SUBAPPLICATION Uebung_072c (* GBSD auf UT ausgeben *)
  (* Standard: 61499-2 *)
  (* Version 1.0, 2023-10-23, franz *)
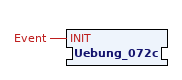
  EVENT_INPUT
    INIT;
  END_EVENT
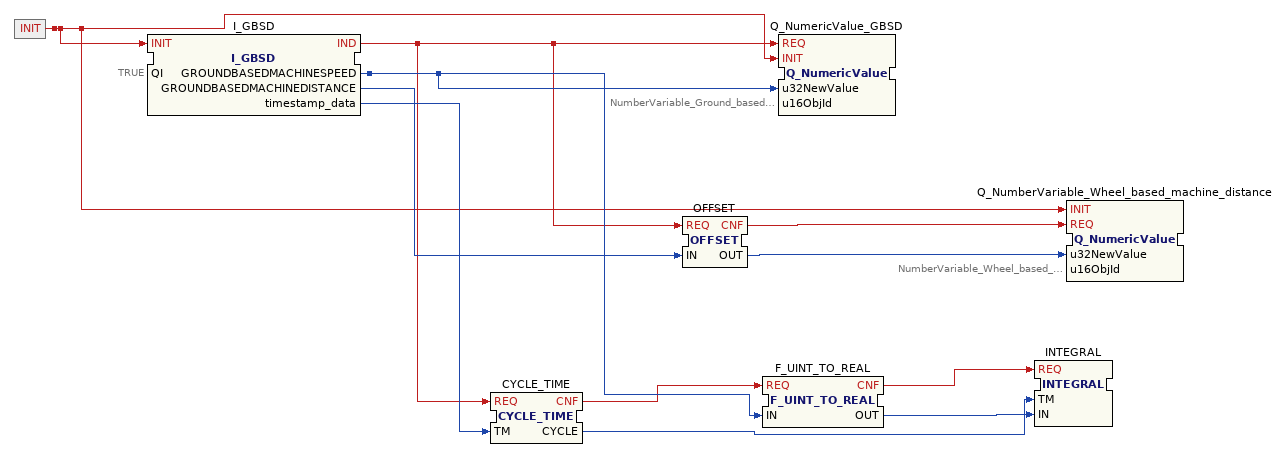
  FBS
    I_GBSD : I_GBSD(QI := TRUE);
    Q_NumericValue_GBSD : Q_NumericValue(u16ObjId := NumberVariable_Ground_based_machine_speed);
    Q_NumberVariable_Wheel_based_machine_distance : Q_NumericValue(u16ObjId := NumberVariable_Wheel_based_machine_distance);
    INTEGRAL : utils::math::INTEGRAL;
    OFFSET : utils::math::OFFSET;
    CYCLE_TIME : utils::timing::CYCLE_TIME;
    F_UINT_TO_REAL : F_UINT_TO_REAL;
  END_FBS
  EVENT_CONNECTIONS
    INIT TO I_GBSD.INIT;
    I_GBSD.IND TO Q_NumericValue_GBSD.REQ;
    INIT TO Q_NumericValue_GBSD.INIT;
    INIT TO Q_NumberVariable_Wheel_based_machine_distance.INIT;
    I_GBSD.IND TO OFFSET.REQ;
    OFFSET.CNF TO Q_NumberVariable_Wheel_based_machine_distance.REQ;
    I_GBSD.IND TO CYCLE_TIME.REQ;
    CYCLE_TIME.CNF TO F_UINT_TO_REAL.REQ;
    F_UINT_TO_REAL.CNF TO INTEGRAL.REQ;
  END_CONNECTIONS
  DATA_CONNECTIONS
    I_GBSD.GROUNDBASEDMACHINESPEED TO Q_NumericValue_GBSD.u32NewValue;
    I_GBSD.GROUNDBASEDMACHINEDISTANCE TO OFFSET.IN;
    OFFSET.OUT TO Q_NumberVariable_Wheel_based_machine_distance.u32NewValue;
    I_GBSD.timestamp_data TO CYCLE_TIME.TM;
    CYCLE_TIME.CYCLE TO INTEGRAL.TM;
    F_UINT_TO_REAL.OUT TO INTEGRAL.IN;
    I_GBSD.GROUNDBASEDMACHINESPEED TO F_UINT_TO_REAL.IN;
  END_CONNECTIONS
END_SUBAPPLICATION
